FUNCTION_BLOCK fb_test_xmeas_simulated


VAR
	
	// data acquitistion from IO blocks
	xmeas_acquire: fb_xmeas_acquire;

	// Molar Percent G control loop
	//pct_g_dpi: fb_discrete_pi		  := (kc:=1, ti:=0.001/60, Ts:=g_Ts_base, hi :=100, lo:=0, x0:=Eadj_0);
	
	// production rate control loop
	prod_rate_loop: fb_prod_rate_ctrl := (kc:=3.2, ti:=120/60, ts:=g_Ts_base, x0:=0, hi:=30, lo:=0);	
	
	// feed ratio control loop
	feed_ratio_ctrl: fb_feed_ratio_ctrl;
	
	// process levels/invetory controller
	level_ctrl: fb_level_ctrl;
		
	// product comnposition controller
	prod_comp_ctrl: fb_prod_comp_ctrl;
	
	// A & C ratio controller
	ac_ratio_ctrl: fb_ac_ratio_ctrl;
	
	// temperature controller
	temp_ctrl: fb_temp_ctrl;
	
	// simulated measurements for debug
	xmeas_simulated: fb_xmeas_simulated;
END_VAR

VAR_INPUT
	
END_VAR

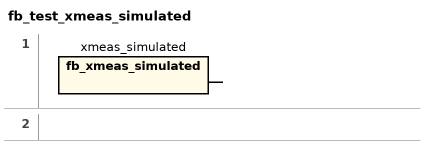
// NETWORK 1
//   xmeas_simulated: simulated measurements for debug
xmeas_simulated(); // fb_xmeas_simulated

// NETWORK 2

END_FUNCTION_BLOCK

(* stored: Version 1.1.0.1, ProductVersion 3.1.0.26
   POU fb_test_xmeas_simulated: Id {b0de2ca6-0986-47af-b383-b23e537ead25} *)
